FUNCTION_BLOCK T_RemoveComponentAtIndexRemovesItem EXTENDS T_UnitTestBase
VAR
END_VAR

TestFinished();

END_FUNCTION_BLOCK

(* stored: Version 1.1.0.1, ProductVersion 3.1.4024.12
   POU T_RemoveComponentAtIndexRemovesItem: Id {a5ac6aae-d815-4031-8abd-dd6bd35c8542}, SpecialFunc None *)
